(* IEC 61131-3 sources: ICSQuartz/benchmarks/icsfuzz_oob_1_arr_6/src, 1 file *)

(* ---- program.st ---- *)
PROGRAM PLC_PRG
VAR
	input1 AT %IW1:WORD;
	output1 AT %QW1:WORD;
	in_addr: DWORD;
	// arr_6: arr_6;
END_VAR
output1 := arr_6(input1);
END_PROGRAM

FUNCTION arr_6 : WORD

VAR_INPUT
	input1: WORD;
END_VAR

VAR
	array1: ARRAY [0 .. 100] OF WORD;
	index1: WORD;
	index2: WORD;
	load_val: WORD;
	iter: DINT;
	cond: WORD;
END_VAR

load_val := 16#DEAD;

index1 := input1/256 + 32;
index2 := input1/512 + 67;

cond := input1/256;

// TODO - verify this
// arr_4 := index1;

FOR iter := 0 TO 100 BY 1 DO
	IF iter < index1 THEN
		// Manual throw
		// IF index1 > 100 THEN
		// 	index1 := 100000;
		// END_IF
		array1[index1] := load_val;
	ELSE
		// Manual throw
		// IF index1 > 100 THEN
		// 	index1 := 100000;
		// END_IF
		array1[index2] := load_val;
	END_IF
END_FOR

arr_6 := index1;
END_FUNCTION
